// TIA Portal V18 export
DATA_BLOCK "CMMS_Z1_FHPP_CTRL_DB"   // DB70
AUTHOR : FESTO
FAMILY : E-DRIVE
VERSION : 5.1
// stored: AutoNumber true, DBAccessibleFromOPCUA true, InstanceOfName FHPP_CTRL, InstanceOfType FB
"FHPP_CTRL"
   // VAR_INPUT
   //    EnableDrive : Bool;
   //    Stop : Bool;
   //    Halt : Bool;
   //    Brake : Bool;
   //    ResetFault : Bool;
   //    HMIAccessLocked : Bool;
   //    OPM : Int;
   //    StartTask : Bool;
   //    StartHoming : Bool;
   //    JogPos : Bool;
   //    JogNeg : Bool;
   //    TeachActValue : Bool;
   //    ClearRemPos : Bool;
   //    Relative : Bool;
   //    DeactivateStrokeLimit : Bool;
   //    ExecuteFunction : Bool;
   //    RecordNo : Int;
   //    SetFunctionNumber : Int;
   //    SetFunctionGroup : Int;
   //    SetValueVelocity : DInt;
   //    SetValuePosition : DInt;
   //    SetValueForceRamp : DInt;
   //    SetValueForce : DInt;
   //    SetValueRotRamp : DInt;
   //    SetValueRotSpeed : DInt;
   // END_VAR
   // VAR_OUTPUT
   //    DriveEnabled : Bool;
   //    Ready : Bool;
   //    Warning : Bool;
   //    Fault : Bool;
   //    SupplyVoltPresent : Bool;
   //    ControlFCT_HMI : Bool;
   //    StateOPM : Int;
   //    HaltNotActive : Bool;
   //    AckStart : Bool;
   //    MC : Bool;
   //    AckTeach : Bool;
   //    DriveMoving : Bool;
   //    DragError : Bool;
   //    StandStillControl : Bool;
   //    HomingValid : Bool;
   //    ActualRecordNo : Int;
   //    RC1 : Bool;
   //    RCC : Bool;
   //    VelocityLimitReached : Bool;
   //    StrokeLimitReached : Bool;
   //    FunctionIsActive : Bool;
   //    ActualFunctionNumber : Int;
   //    ActualFunctionGroup : Int;
   //    ActualPosition : DInt;
   //    ActualVelocity : DInt;
   //    ActualForce : DInt;
   //    ActualRotRamp : DInt;
   //    ActualRotSpeed : DInt;
   // END_VAR
   // VAR_IN_OUT
   //    FML_REF : "DT_FML_REF";
   // END_VAR
   // VAR
   //    Converted_BYTE5_8_IN : DInt;
   //    Converted_BYTE5_8_OUT : DInt;
   //    OperationModeB1 : Bool;
   //    OperationModeB2 : Bool;
   //    ControlModeB1 : Bool;
   //    ControlModeB2 : Bool;
   //    ContinuousMode : Bool;
   //    StateOperationModeB1 : Bool;
   //    StateOperationModeB2 : Bool;
   //    StateControlModeB1 : Bool;
   //    StateControlModeB2 : Bool;
   //    StateContinuousMode : Bool;
   // END_VAR
BEGIN
END_DATA_BLOCK
